Universal Robots PolyScope program: recogeHuevos.urp

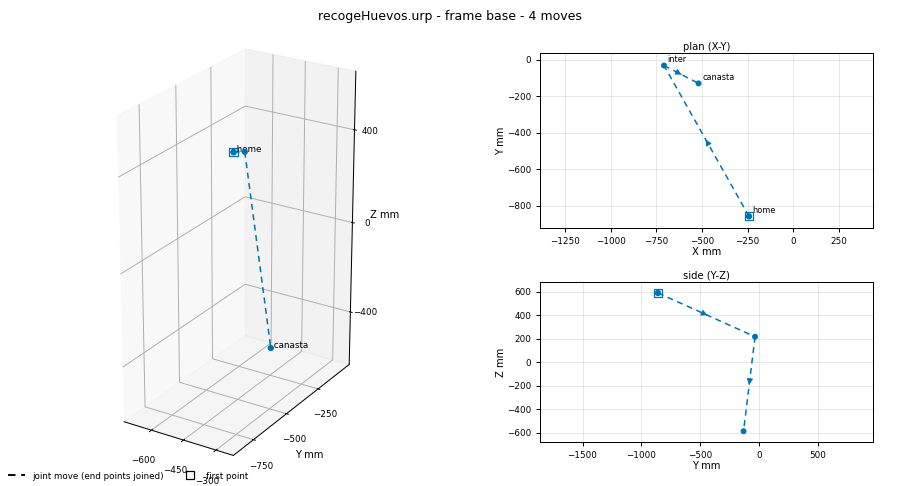
[picture p0: tool path of recogeHuevos.urp in frame base, 4 of 4 moves have a stored position in this frame; points joined in program order, loops and branches not executed]
Program recogeHuevos (installation=default directory=/programs/usbdisk/reto createdIn=5.13.0 lastSavedIn=5.13.0 robotSerialNumber=20205500280)
Calibrated DH parameters: a=[0.000126, -0.227628, -0.392536, 0.000072, 0.000053, 0]; d=[0.16267, 78.773992, -78.210517, -0.430145, 0.099656, 0.099678]; alpha=[1.568545, -0.004566, 0.00572, 1.569931, -1.57104, 0]; deltaTheta=[0, -1.006608, 7.298003, -0.008206, 0.000004, 0]
InitVariablesNode
Robot Program (runOnlyOnce=false)
  MoveJ speed 60 deg/s, acceleration 80 deg/s^2 (useActiveTCP=true) feature=Base
    Waypoint home: TCP in base x=-242.78 y=-857.838 z=589.961 mm, rx=-0.5599 ry=-1.8727 rz=1.9411 rad; joints [70.139, -63.013, 42.403, 18.907, 102.438, 0.999] deg; TCP offset x=0 y=0 z=234.35 mm, rx=0 ry=0 rz=-3.1416 rad
  init := 0
  var_3 := 0
  URCap Subscribe Topic (ros_as_a_service, FZI Research Center for Information Technology) dataModel(MASTER_NAME=default, MASTER=192.168.0.229, PORT=9090, MSG=/my_topic/int, MSG_LAYOUT_Data=[{"fieldnames":["data"],"fieldtypes":["int32"],"examples":["0"],"fieldarraylen":[-1],"constvalues":[],"constnames":[],"type":"std_msgs/Int32"}], MSG_VALUE_Data={"data":{"-+useVarNum+-":"init"}})
  Switch expression=init
    Case (caseValue=1)
      MoveJ speed 60 deg/s, acceleration 80 deg/s^2 (useActiveTCP=true) feature=Base
        Waypoint huevo1: TCP in base x=-242.727 y=-857.899 z=589.927 mm, rx=-0.5599 ry=-1.8727 rz=1.9412 rad; joints [70.143, -63.008, 42.4, 18.903, 102.438, 1.001] deg; TCP offset x=0 y=0 z=234.35 mm, rx=0 ry=0 rz=-3.1416 rad
        huevo11 := huevo1
    Case (caseValue=2)
      MoveJ speed 60 deg/s, acceleration 80 deg/s^2 (useActiveTCP=true) feature=Base
        Waypoint inter: TCP in base x=-708.33 y=-31.819 z=217.607 mm, rx=-1.9455 ry=-1.7364 rz=0.276 rad; joints [-2.43, -55.509, 50.085, 65.759, 102.419, 1.013] deg
        Waypoint canasta: TCP in base x=-519.086 y=-129.593 z=-586.57 mm, rx=-2.2239 ry=-2.1926 rz=0.0004 rad; joints [-0.241, 10.034, 50.044, 29.182, 90.893, 0.995] deg
  Wait Sleep waitTime=1
  URCap Publish Topic (ros_as_a_service, FZI Research Center for Information Technology) dataModel(MASTER_NAME=default, MASTER=192.168.0.229, PORT=9090, MSG=/my_topic/string, MSG_LAYOUT_Data=[{"fieldnames":["data"],"fieldtypes":["string"],"examples":[""],"fieldarraylen":[-1],"constvalues":[],"constnames":[],"type":"std_msgs/String"}], MSG_VALUE_Data={"data":{"-+useVar+-":"huevo11"}})
